(* CoDeSys 2.3 export: CILINDRO_DOBLE.EXP *)

(* Data type *)
TYPE Cilindro_Doble :
STRUCT
	Valvula                       : EV_Doble;
	Sensor_Avance       : Sensor_Magnetico;
	Sensor_Retroceso : Sensor_Magnetico;
END_STRUCT
END_TYPE
